// Mitsubishi GX Works2 project: inverter-3   PLC: Q03UDV

PROGRAM MAIN
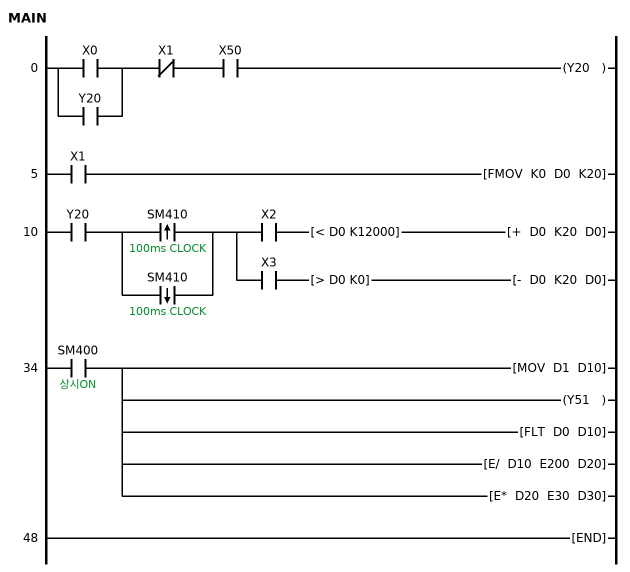
0     LD      X0
      OR      Y20
      ANI     X1
      AND     X50
      OUT     Y20
5     LD      X1
      FMOV    K0 D0 K20
10    LD      Y20
      LDP     SM410  ; 100ms CLOCK
      ORF     SM410  ; 100ms CLOCK
      ANB
      MPS
      AND     X2
      AND<    D0 K12000
      +       D0 K20 D0
      MPP
      AND     X3
      AND>    D0 K0
      -       D0 K20 D0
34    LD      SM400  ; 상시ON
      MOV     D1 D10
      OUT     Y51
      FLT     D0 D10
      E/      D10 E200 D20
      E*      D20 E30 D30
48    END
END_PROGRAM
